{attribute 'qualified_only'}
{attribute 'strict'}
{attribute 'to_string'}
TYPE E_HE_SolidAttenuatorCalculationMode :
(
    FLOOR := 0,
    CEILING := 1,
    WITHIN_TOLERANCE := 2
) INT;
END_TYPE

(* stored: Version 1.1.0.1
   DUT E_HE_SolidAttenuatorCalculationMode: Id {047ac3c6-40e5-4417-84dc-5d1b4583e4de} *)
